// TIA Portal V17 export
// export: Created 2023-12-22T15:28:30.1298148Z, ExportSetting WithDefaults, DisplayName Totally Integrated Automation Portal, DisplayVersion V17, DisplayName TIA Portal Openness, DisplayVersion V17, DisplayName TIA Portal Version Control Interface, DisplayVersion V17, DisplayName STEP 7 Professional, DisplayVersion V17, DisplayName STEP 7 Safety, DisplayVersion V17, DisplayName WinCC Advanced, DisplayVersion V17
FUNCTION_BLOCK "PID_ex"   // FB99, LAD
{ S7_Optimized_Access := 'FALSE' }
VERSION : 0.1
// stored: AutoNumber false, IsIECCheckEnabled false, SetENOAutomatically false, UDAEnableTagReadback false
   VAR_INPUT
      Start : Bool;
      SP_A : Real;   // Уставка
      Value : Real;   // Показания датчика
   END_VAR
   VAR_OUTPUT
      PWM : Bool;   // ШИМ-выход ПИД-регулятора
      Result : Real;   // Управляющее воздействие
   END_VAR
   VAR DB_SPECIFIC
      CMD { S7_SetPoint := 'True'} : "CMD";
      SP_M : Real;
      SP : Real;
      x { S7_SetPoint := 'True'} : Real := 1.0;   // Поправка уставки и датчика
      SP_x : Real;   // Домноженная уставка
      Value_x : Real;   // Домноженный датчик
      Buffer : Real;   // Промежуточное значение
      PID_Output : Real;   // Выход ПИД-регулятора
      PID_Hand : Real;   // Ручное задание выхода ПИД-регулятора
      Sys : Struct   // Системные параметры
         Err_Ack : Bool;   // Подтверждение аварии
         Alm_SP_H : Bool;   // Авария уставки - превышение
         Alm_SP_L : Bool;   // Авария уставки - занижение
         Alm_In_H : Bool;   // Авария датчика - превышение
         Alm_In_L : Bool;   // Авария датчика - занижение
         Activate : Bool;   // Активировать ПИД
         Error_code : DWord;   // Код аварии
         Warning_code : DWord;   // Код предупреждения
         "Type" : Int := 1;   // Режим работы
         State : Int;   // Состояние
         Mode : Int := 3;   // Режим
      END_STRUCT;
      Settings : Struct   // Рабочие параметры
         SP_P { S7_SetPoint := 'True'} : Real := 1.5;   // Коэффициент пропорциональности
         SP_Ti { S7_SetPoint := 'True'} : Real := 150.0;   // Время интегрирования
         SP_Td { S7_SetPoint := 'True'} : Real;   // Время дифференцирования
         SP_Cycle { S7_SetPoint := 'True'} : Real := 0.2;   // Время цикла
         Max_SP { S7_SetPoint := 'True'} : Real := 500.0;   // Максимальное значение уставки
         Min_SP { S7_SetPoint := 'True'} : Real := -500.0;   // Минимальное значение уставки
         Max_in { S7_SetPoint := 'True'} : Real := 500.0;   // Максимальное значение датчика
         Min_in { S7_SetPoint := 'True'} : Real := -500.0;   // Минимальное значение датчика
         Max_out { S7_SetPoint := 'True'} : Real := 100.0;   // Максимальное значение выхода
         Min_out { S7_SetPoint := 'True'} : Real := 0.0;   // Минимальное значение выхода
         DeadBand { S7_SetPoint := 'True'} : Real := 1.0;   // Мёртвая зона
         Max : Real;   // Верняя граница мёртвой зоны
         Min : Real;   // Нижняя граница мёртвой зоны
      END_STRUCT;
   END_VAR
   VAR
      PID { S7_SetPoint := 'True'} : PID_Compact;   // ПИД
      Converter : "Converter";   // Конвертер выхода
      Conveter_Back : "Converter";   // Конвертер Hand_SP в 0..100
      C { S7_SetPoint := 'True'} : "Time_R";   // Частота вызова ПИД на обработку
   END_VAR
   VAR DB_SPECIFIC
      pos : Array[0..15] of Bool;
   END_VAR
   VAR_TEMP
      x0 : Real;
   END_VAR
   // CMD.Start_A := true;
   // Converter.Max_In := 100.0;
   // Conveter_Back.Max_Out := 100.0;
   VAR_TEMP   // added for the SCL form of the ladder/FBD networks
      _w1 : Bool;
      _w2 : Bool;
   END_VAR
BEGIN

REGION Network 1: Сброс ПИД
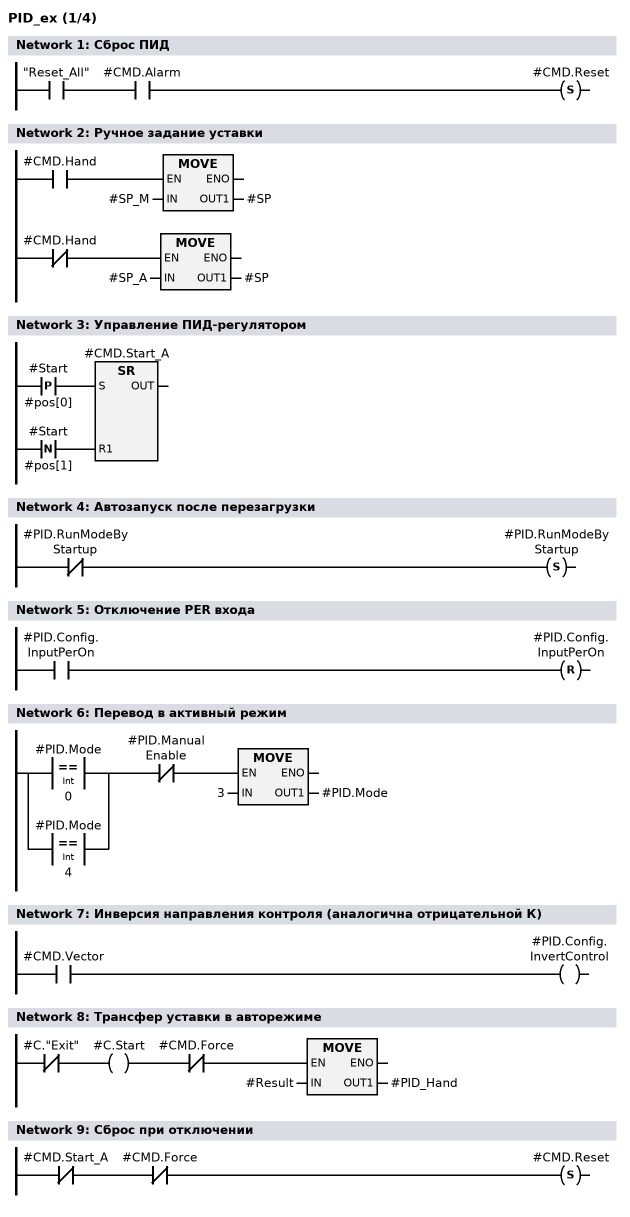
   RUNG wire#powerrail
      Contact( "Reset_All" )
      Contact( #CMD.Alarm )
      S_Coil( #CMD.Reset )
   END_RUNG
   // the same network as SCL:
   IF "Reset_All" AND #CMD.Alarm THEN #CMD.Reset := TRUE; END_IF;
END_REGION

REGION Network 2: Ручное задание уставки
   RUNG wire#powerrail
      Contact( #CMD.Hand )
      Move(in := #SP_M, out1 => #SP)
   END_RUNG
   RUNG wire#powerrail
      I_Contact( #CMD.Hand )
      Move(in := #SP_A, out1 => #SP)
   END_RUNG
   // the same network as SCL:
   IF #CMD.Hand THEN #SP := #SP_M; END_IF;
   IF NOT #CMD.Hand THEN #SP := #SP_A; END_IF;
END_REGION

REGION Network 3: Управление ПИД-регулятором
   RUNG wire#powerrail
      P_Contact(operand := #Start, bit := #pos[0])
      S_SR(operand := #CMD.Start_A, r1 := wire#w1)
   END_RUNG
   RUNG wire#powerrail
      N_Contact(operand := #Start, bit := #pos[1])
   END_RUNG wire#w1
   // the same network as SCL:
   #_w1 := #Start AND NOT #pos[0];   // rising edge of #Start
   #pos[0] := #Start;
   #_w2 := NOT #Start AND #pos[1];   // falling edge of #Start
   #pos[1] := #Start;
   IF #_w1 THEN
       #CMD.Start_A := TRUE;   // SR flip-flop
   END_IF;
   IF #_w2 THEN #CMD.Start_A := FALSE; END_IF;
END_REGION

REGION Network 4: Автозапуск после перезагрузки
   RUNG wire#powerrail
      I_Contact( #PID.RunModeByStartup )
      S_Coil( #PID.RunModeByStartup )
   END_RUNG
   // the same network as SCL:
   IF NOT #PID.RunModeByStartup THEN #PID.RunModeByStartup := TRUE; END_IF;
END_REGION

REGION Network 5: Отключение PER входа
   RUNG wire#powerrail
      Contact( #PID.Config.InputPerOn )
      R_Coil( #PID.Config.InputPerOn )
   END_RUNG
   // the same network as SCL:
   IF #PID.Config.InputPerOn THEN #PID.Config.InputPerOn := FALSE; END_IF;
END_REGION

REGION Network 6: Перевод в активный режим
   RUNG wire#powerrail
      { S7_Templates := "SrcType := Int" } EQ_Contact(in1 := #PID.Mode, in2 := 0)
      wire#w1
      I_Contact( #PID.ManualEnable )
      { S7_GenerateENO := "TRUE" } Move(in := 3, out1 => #PID.Mode)
   END_RUNG
   RUNG wire#powerrail
      { S7_Templates := "SrcType := Int" } EQ_Contact(in1 := #PID.Mode, in2 := 4)
   END_RUNG wire#w1
   // the same network as SCL:
   IF ((#PID.Mode = 0) OR (#PID.Mode = 4)) AND NOT #PID.ManualEnable THEN #PID.Mode := 3; END_IF;
END_REGION

REGION Network 7: Инверсия направления контроля (аналогична отрицательной К)
   RUNG wire#powerrail
      Contact( #CMD.Vector )
      Coil( #PID.Config.InvertControl )
   END_RUNG
   // the same network as SCL:
   #PID.Config.InvertControl := #CMD.Vector;
END_REGION

REGION Network 8: Трансфер уставки в авторежиме
   RUNG wire#powerrail
      I_Contact( #C."Exit" )
      Coil( #C.Start )
      I_Contact( #CMD.Force )
      Move(in := #Result, out1 => #PID_Hand)
   END_RUNG
   // the same network as SCL:
   #C.Start := NOT #C."Exit";
   IF NOT #C."Exit" AND NOT #CMD.Force THEN #PID_Hand := #Result; END_IF;
END_REGION

REGION Network 9: Сброс при отключении
   RUNG wire#powerrail
      I_Contact( #CMD.Start_A )
      I_Contact( #CMD.Force )
      S_Coil( #CMD.Reset )
   END_RUNG
   // the same network as SCL:
   IF NOT #CMD.Start_A AND NOT #CMD.Force THEN #CMD.Reset := TRUE; END_IF;
END_REGION

REGION Network 10: Активация после смены режима
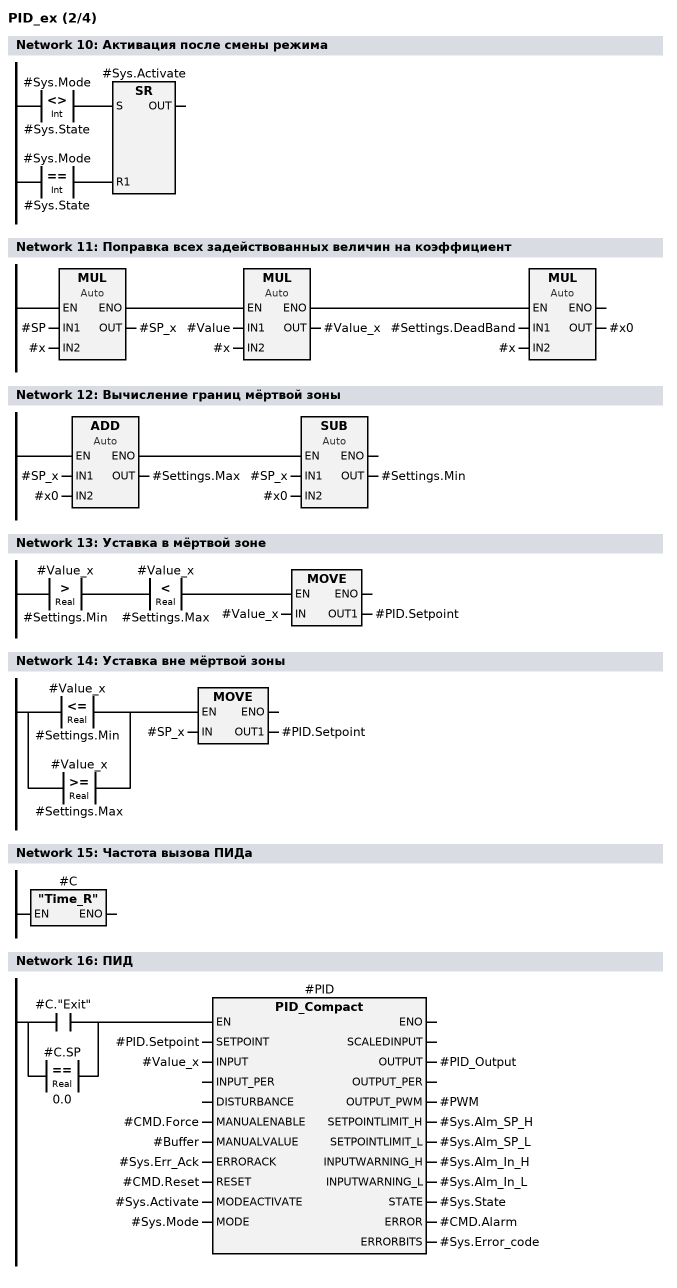
   RUNG wire#powerrail
      { S7_Templates := "SrcType := Int" } NE_Contact(in1 := #Sys.Mode, in2 := #Sys.State)
      S_SR(operand := #Sys.Activate, r1 := wire#w1)
   END_RUNG
   RUNG wire#powerrail
      { S7_Templates := "SrcType := Int" } EQ_Contact(in1 := #Sys.Mode, in2 := #Sys.State)
   END_RUNG wire#w1
   // the same network as SCL:
   IF #Sys.Mode <> #Sys.State THEN
       #Sys.Activate := TRUE;   // SR flip-flop
   END_IF;
   IF #Sys.Mode = #Sys.State THEN #Sys.Activate := FALSE; END_IF;
END_REGION

REGION Network 11: Поправка всех задействованных величин на коэффициент
   RUNG wire#powerrail
      Mul(in1 := #SP, in2 := #x, out => #SP_x)
      Mul(in1 := #Value, in2 := #x, out => #Value_x)
      Mul(in1 := #Settings.DeadBand, in2 := #x, out => #x0)
   END_RUNG
   // the same network as SCL:
   #SP_x := #SP * #x;
   #Value_x := #Value * #x;
   #x0 := #Settings.DeadBand * #x;
END_REGION

REGION Network 12: Вычисление границ мёртвой зоны
   RUNG wire#powerrail
      Add(in1 := #SP_x, in2 := #x0, out => #Settings.Max)
      Sub(in1 := #SP_x, in2 := #x0, out => #Settings.Min)
   END_RUNG
   // the same network as SCL:
   #Settings.Max := #SP_x + #x0;
   #Settings.Min := #SP_x - #x0;
END_REGION

REGION Network 13: Уставка в мёртвой зоне
   RUNG wire#powerrail
      { S7_Templates := "SrcType := Real" } GT_Contact(in1 := #Value_x, in2 := #Settings.Min)
      { S7_Templates := "SrcType := Real" } LT_Contact(in1 := #Value_x, in2 := #Settings.Max)
      Move(in := #Value_x, out1 => #PID.Setpoint)
   END_RUNG
   // the same network as SCL:
   IF (#Value_x > #Settings.Min) AND (#Value_x < #Settings.Max) THEN #PID.Setpoint := #Value_x; END_IF;
END_REGION

REGION Network 14: Уставка вне мёртвой зоны
   RUNG wire#powerrail
      { S7_Templates := "SrcType := Real" } LE_Contact(in1 := #Value_x, in2 := #Settings.Min)
      wire#w1
      Move(in := #SP_x, out1 => #PID.Setpoint)
   END_RUNG
   RUNG wire#powerrail
      { S7_Templates := "SrcType := Real" } GE_Contact(in1 := #Value_x, in2 := #Settings.Max)
   END_RUNG wire#w1
   // the same network as SCL:
   IF (#Value_x <= #Settings.Min) OR (#Value_x >= #Settings.Max) THEN #PID.Setpoint := #SP_x; END_IF;
END_REGION

REGION Network 15: Частота вызова ПИДа
   RUNG wire#powerrail
      #C()
   END_RUNG
   // the same network as SCL:
   #C();   // "Time_R"
END_REGION

REGION Network 16: ПИД
   RUNG wire#powerrail
      Contact( #C."Exit" )
      wire#w1
      #PID.PID_Compact(Setpoint := #PID.Setpoint, Input := #Value_x, Input_PER :=, Disturbance :=, ManualEnable := #CMD.Force, ManualValue := #Buffer, ErrorAck := #Sys.Err_Ack, Reset := #CMD.Reset, ModeActivate := #Sys.Activate, Mode := #Sys.Mode, ScaledInput =>, Output => #PID_Output, Output_PER =>, Output_PWM => #PWM, SetpointLimit_H => #Sys.Alm_SP_H, SetpointLimit_L => #Sys.Alm_SP_L, InputWarning_H => #Sys.Alm_In_H, InputWarning_L => #Sys.Alm_In_L, State => #Sys.State, Error => #CMD.Alarm, ErrorBits => #Sys.Error_code)
   END_RUNG
   RUNG wire#powerrail
      { S7_Templates := "SrcType := Real" } EQ_Contact(in1 := #C.SP, in2 := 0.0)
   END_RUNG wire#w1
   // the same network as SCL:
   IF #C."Exit" OR (#C.SP = 0.0) THEN
       #PID(Setpoint := #PID.Setpoint,   // PID_Compact
            Input := #Value_x,
            ManualEnable := #CMD.Force,
            ManualValue := #Buffer,
            ErrorAck := #Sys.Err_Ack,
            Reset := #CMD.Reset,
            ModeActivate := #Sys.Activate,
            Mode := #Sys.Mode,
            Output => #PID_Output,
            Output_PWM => #PWM,
            SetpointLimit_H => #Sys.Alm_SP_H,
            SetpointLimit_L => #Sys.Alm_SP_L,
            InputWarning_H => #Sys.Alm_In_H,
            InputWarning_L => #Sys.Alm_In_L,
            State => #Sys.State,
            Error => #CMD.Alarm,
            ErrorBits => #Sys.Error_code);
   END_IF;
END_REGION

REGION Network 17: Обратное масштабирование в ручном режиме
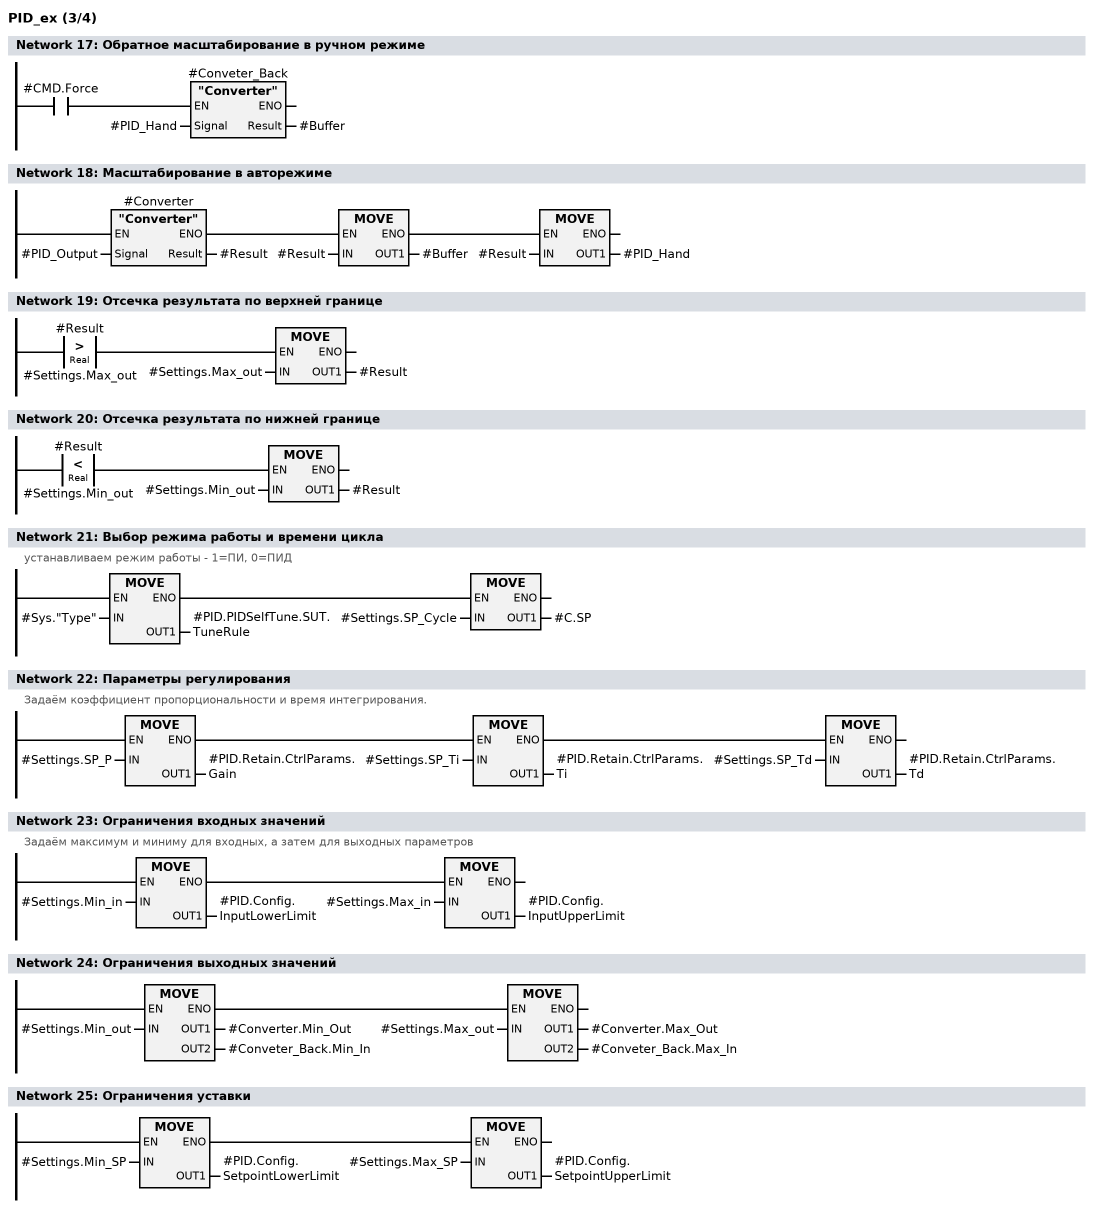
   RUNG wire#powerrail
      Contact( #CMD.Force )
      #Conveter_Back(Signal := #PID_Hand, Result => #Buffer)
   END_RUNG
   // the same network as SCL:
   IF #CMD.Force THEN
       #Conveter_Back(Signal := #PID_Hand, Result => #Buffer);   // "Converter"
   END_IF;
END_REGION

REGION Network 18: Масштабирование в авторежиме
   RUNG wire#powerrail
      #Converter(Signal := #PID_Output, Result => #Result)
      { S7_GenerateENO := "TRUE" } Move(in := #Result, out1 => #Buffer)
      { S7_GenerateENO := "TRUE" } Move(in := #Result, out1 => #PID_Hand)
   END_RUNG
   // the same network as SCL:
   // ENO of a box is taken as its EN; it also drops when the box reports an error
   #Converter(Signal := #PID_Output, Result => #Result, ENO => #_w1);   // "Converter"
   IF #_w1 THEN
       #Buffer := #Result;
       #PID_Hand := #Result;
   END_IF;
END_REGION

REGION Network 19: Отсечка результата по верхней границе
   RUNG wire#powerrail
      { S7_Templates := "SrcType := Real" } GT_Contact(in1 := #Result, in2 := #Settings.Max_out)
      Move(in := #Settings.Max_out, out1 => #Result)
   END_RUNG
   // the same network as SCL:
   IF #Result > #Settings.Max_out THEN #Result := #Settings.Max_out; END_IF;
END_REGION

REGION Network 20: Отсечка результата по нижней границе
   RUNG wire#powerrail
      { S7_Templates := "SrcType := Real" } LT_Contact(in1 := #Result, in2 := #Settings.Min_out)
      Move(in := #Settings.Min_out, out1 => #Result)
   END_RUNG
   // the same network as SCL:
   IF #Result < #Settings.Min_out THEN #Result := #Settings.Min_out; END_IF;
END_REGION

REGION Network 21: Выбор режима работы и времени цикла
   // устанавливаем режим работы - 1=ПИ, 0=ПИД
   RUNG wire#powerrail
      { S7_GenerateENO := "TRUE" } Move(in := #Sys."Type", out1 => #PID.PIDSelfTune.SUT.TuneRule)
      { S7_GenerateENO := "TRUE" } Move(in := #Settings.SP_Cycle, out1 => #C.SP)
   END_RUNG
   // the same network as SCL:
   // ENO of a box is taken as its EN; it also drops when the box reports an error
   #PID.PIDSelfTune.SUT.TuneRule := #Sys."Type";
   #C.SP := #Settings.SP_Cycle;
END_REGION

REGION Network 22: Параметры регулирования
   // Задаём коэффициент пропорциональности и время интегрирования.
   RUNG wire#powerrail
      { S7_GenerateENO := "TRUE" } Move(in := #Settings.SP_P, out1 => #PID.Retain.CtrlParams.Gain)
      { S7_GenerateENO := "TRUE" } Move(in := #Settings.SP_Ti, out1 => #PID.Retain.CtrlParams.Ti)
      { S7_GenerateENO := "TRUE" } Move(in := #Settings.SP_Td, out1 => #PID.Retain.CtrlParams.Td)
   END_RUNG
   // the same network as SCL:
   // ENO of a box is taken as its EN; it also drops when the box reports an error
   #PID.Retain.CtrlParams.Gain := #Settings.SP_P;
   #PID.Retain.CtrlParams.Ti := #Settings.SP_Ti;
   #PID.Retain.CtrlParams.Td := #Settings.SP_Td;
END_REGION

REGION Network 23: Ограничения входных значений
   // Задаём максимум и миниму для входных, а затем для выходных параметров
   RUNG wire#powerrail
      { S7_GenerateENO := "TRUE" } Move(in := #Settings.Min_in, out1 => #PID.Config.InputLowerLimit)
      { S7_GenerateENO := "TRUE" } Move(in := #Settings.Max_in, out1 => #PID.Config.InputUpperLimit)
   END_RUNG
   // the same network as SCL:
   // ENO of a box is taken as its EN; it also drops when the box reports an error
   #PID.Config.InputLowerLimit := #Settings.Min_in;
   #PID.Config.InputUpperLimit := #Settings.Max_in;
END_REGION

REGION Network 24: Ограничения выходных значений
   RUNG wire#powerrail
      { S7_GenerateENO := "TRUE" } Move(in := #Settings.Min_out, out1 => #Converter.Min_Out, out2 => #Conveter_Back.Min_In)
      { S7_GenerateENO := "TRUE" } Move(in := #Settings.Max_out, out1 => #Converter.Max_Out, out2 => #Conveter_Back.Max_In)
   END_RUNG
   // the same network as SCL:
   // ENO of a box is taken as its EN; it also drops when the box reports an error
   #Converter.Min_Out := #Settings.Min_out;
   #Conveter_Back.Min_In := #Settings.Min_out;
   #Converter.Max_Out := #Settings.Max_out;
   #Conveter_Back.Max_In := #Settings.Max_out;
END_REGION

REGION Network 25: Ограничения уставки
   RUNG wire#powerrail
      { S7_GenerateENO := "TRUE" } Move(in := #Settings.Min_SP, out1 => #PID.Config.SetpointLowerLimit)
      { S7_GenerateENO := "TRUE" } Move(in := #Settings.Max_SP, out1 => #PID.Config.SetpointUpperLimit)
   END_RUNG
   // the same network as SCL:
   // ENO of a box is taken as its EN; it also drops when the box reports an error
   #PID.Config.SetpointLowerLimit := #Settings.Min_SP;
   #PID.Config.SetpointUpperLimit := #Settings.Max_SP;
END_REGION

REGION Network 26: Сброс сброса
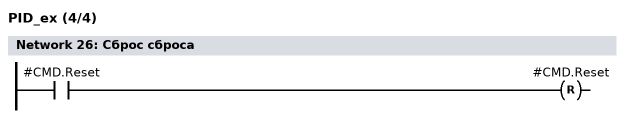
   RUNG wire#powerrail
      Contact( #CMD.Reset )
      R_Coil( #CMD.Reset )
   END_RUNG
   // the same network as SCL:
   IF #CMD.Reset THEN #CMD.Reset := FALSE; END_IF;
END_REGION
END_FUNCTION_BLOCK
